// TIA Portal project "Delta_191206" (V15)

(* hardware
DEVICE "S7-1200 station_1"  S7-1200 Station
   slot 0: "Rack_0"  S7-1200 Rack  Rack  V1.0
   slot 1: "PLC_1"  CPU 1215C DC/DC/DC  6ES7 215-1AG40-0XB0  V4.2
   slot 2: "DQ 16x24VDC_1"  6ES7 222-1BH30-0XB0  V1.0
DEVICE "PC station"  SIMATIC PC station
   slot 0: "PC station"  Rail  SIMATIC PC-Station  V1.0
      slot 125: "Stationmanager"  Station_Manager  V6.0.4
   slot 1: "IE general"  IE General  IE_CP  V8.2.0
   slot 2: "OPC Server_1"  OPC Server  OPC Server  V8.2.0
*)

// ===== PLC "PLC_1"  CPU 1215C DC/DC/DC =====

VAR_GLOBAL   // PLC tag table "Default tag table"
   "start" AT %I0.2 : Bool;
   "stop" AT %I0.3 : Bool;
   "AX_1_Homing switch" AT %I1.2 : Bool;
   "Ready" AT %I0.5 : Bool;
   "Emergency_Stop" AT %I0.7 : Bool;
   "AX_2_Homing switch" AT %I1.1 : Bool;
   "Home" AT %I0.4 : Bool;
   "AX_3_Homing switch" AT %I1.3 : Bool;
   "Tag_13" AT %I0.0 : Bool;
   "Tag_14" AT %I0.1 : Bool;
   "AX_1_Pulse" AT %Q0.0 : Bool;
   "AX_1_Direction" AT %Q0.3 : Bool;
   "AX_1_DriveEnable" AT %Q0.6 : Bool;
   "AX_2_Pulse" AT %Q0.1 : Bool;
   "AX_2_Direction" AT %Q0.4 : Bool;
   "AX_2_DriveEnable" AT %Q0.7 : Bool;
   "AX_3_Direction" AT %Q0.5 : Bool;
   "AX_3_Pulse" AT %Q0.2 : Bool;
   "AX_3_DriveEnable" AT %Q1.0 : Bool;
   "Sys_Start" AT %M0.0 : Bool;
   "tr_0" AT %M1.0 : Bool;
   "pos_on" AT %M2.0 : Bool;
   "AX_1_done" AT %M3.0 : Bool;
   "AX_2_done" AT %M3.1 : Bool;
   "AX_3_done" AT %M3.2 : Bool;
   "done_1" AT %M3.3 : Bool;
   "done_2" AT %M3.4 : Bool;
   "done_3" AT %M3.5 : Bool;
   "ind" AT %MW4 : Int;
   "tr_1" AT %M1.1 : Bool;
   "tr_3" AT %M1.3 : Bool;
   "tr_4" AT %M1.4 : Bool;
   "tr_5" AT %M1.5 : Bool;
   "tr_6" AT %M1.6 : Bool;
   "Tag_8" AT %M0.1 : Bool;
   "Tag_9" AT %M0.2 : Bool;
   "tr_7" AT %M1.7 : Bool;
   "tr_2" AT %M1.2 : Bool;
   "Tag_3" AT %M2.2 : Bool;
   "Tag_4" AT %M2.1 : Bool;
   "Tag_5" AT %M2.3 : Bool;
   "Tag_6" AT %M2.4 : Bool;
   "home_ypd" AT %M2.5 : Bool;
   "Tag_2" AT %MD6 : Real;
   "Tag_10" AT %MD10 : Real;
   "Tag_11" AT %MD14 : Real;
   "Tag_12" AT %MD20 : Real;
   "Tag_15" AT %M20.0 : Bool;
   "Tag_16" AT %M2.7 : Bool;
   "Tag_17" AT %M20.3 : Bool;
   "Tag_18" AT %M20.4 : Bool;
   "Tag_19" AT %M20.5 : Bool;
   "Tag_20" AT %M20.1 : Bool;
   "Tag_21" AT %M20.2 : Bool;
   "Tag_22" AT %M20.6 : Bool;
   "Tag_23" AT %M20.7 : Bool;
   "Tag_7" AT %M21.0 : Bool;
   "vakum" AT %Q1.1 : Bool;
   "Tag_25" AT %M4.0 : Bool;
   "Tag_26" AT %M22.0 : Bool;
   "Reset" AT %I0.6 : Bool;
   "gui_start" AT %M23.0 : Bool;
   "gui_stop" AT %M23.1 : Bool;
   "gui_homing" AT %M23.2 : Bool;
   "gui_startpackaging" AT %M23.3 : Bool;
   "gui_reset" AT %M23.4 : Bool;
END_VAR

DATA_BLOCK "OPC_DATA"   // DB5
{ S7_Optimized_Access := 'FALSE' }
VERSION : 0.1
   VAR
      x1_pos : Array[0..100] of Real;
      x2_pos : Array[0..100] of Real;
      x3_pos : Array[0..100] of Real;
      x1_vlcty : Array[0..100] of Real;
      x2_vlcty : Array[0..100] of Real;
      x3_vlcty : Array[0..100] of Real;
      manuel_array : Array[0..100] of Int;
      vakum : Array[0..100] of Int;
   END_VAR
BEGIN
   x1_pos[1] := 0.0;
   x1_pos[0] := 0.0;
   x2_pos[0] := 0.0;
   x2_pos[1] := 0.0;
   x3_pos[0] := 0.0;
   x3_pos[1] := 0.0;
   x1_pos[2] := 0.0;
END_DATA_BLOCK

DATA_BLOCK "AX_1"   // DB1, Motion_DB
{ S7_Optimized_Access := 'TRUE' }
AUTHOR : SIMATIC
FAMILY : BasicMC
NAME : TO_PosAx
VERSION : 6.0
// stored: InstanceOfName TO_PositioningAxis
"TO_PositioningAxis"
BEGIN
   // Axis.HomingReferencePointSwitch_AddressCU = %I1.2
   // Axis.EnableOutput_AddressCU = %Q0.6
   // Axis.DirectionOutputEnabledCU = TRUE
   // Axis.OnlinePtoModeCU = 16#0000_0002
   // Axis.SelectedChannel2EnumCU = %Q0.3
   // Axis.SelectedChannel1EnumCU = %Q0.0
   // Pulse.MinDeltaDeltaFrequencyCU = 0.004
   // Pulse.MaxDeltaDeltaFrequencyCU = 1.0E+10
   // Pulse.MinDeltaFrequencyCU = 0.005
   // Pulse.MaxDeltaFrequencyCU = 9.5E+9
   // Pulse.MinFrequencyCU = 1.0
   // Pulse.MaxFrequencyCU = 100000.0
   // Pulse.OutputSourceCU = 16#0000_0000
   // Axis.SelectPTO = 0
END_DATA_BLOCK

DATA_BLOCK "AX_2"   // DB2, Motion_DB
{ S7_Optimized_Access := 'TRUE' }
AUTHOR : SIMATIC
FAMILY : BasicMC
NAME : TO_PosAx
VERSION : 6.0
// stored: InstanceOfName TO_PositioningAxis
"TO_PositioningAxis"
BEGIN
   // Axis.HomingReferencePointSwitch_AddressCU = %I1.1
   // Axis.EnableOutput_AddressCU = %Q0.7
   // Axis.DirectionOutputEnabledCU = TRUE
   // Axis.OnlinePtoModeCU = 16#0000_0002
   // Axis.SelectedChannel2EnumCU = %Q0.4
   // Axis.SelectedChannel1EnumCU = %Q0.1
   // Pulse.MinDeltaDeltaFrequencyCU = 0.004
   // Pulse.MaxDeltaDeltaFrequencyCU = 1.0E+10
   // Pulse.MinDeltaFrequencyCU = 0.005
   // Pulse.MaxDeltaFrequencyCU = 9.5E+9
   // Pulse.MinFrequencyCU = 1.0
   // Pulse.MaxFrequencyCU = 100000.0
   // Pulse.OutputSourceCU = 16#0000_0000
   // Axis.SelectPTO = 1
   // Axis.OnlinePtoIndexCU = 1
END_DATA_BLOCK

DATA_BLOCK "AX_3"   // DB3, Motion_DB
{ S7_Optimized_Access := 'TRUE' }
AUTHOR : SIMATIC
FAMILY : BasicMC
NAME : TO_PosAx
VERSION : 6.0
// stored: InstanceOfName TO_PositioningAxis
"TO_PositioningAxis"
BEGIN
   // Axis.HomingReferencePointSwitch_AddressCU = %I1.3
   // Axis.EnableOutput_AddressCU = %Q1.0
   // Axis.DirectionOutputEnabledCU = TRUE
   // Axis.OnlinePtoModeCU = 16#0000_0002
   // Axis.SelectedChannel2EnumCU = %Q0.5
   // Axis.SelectedChannel1EnumCU = %Q0.2
   // Pulse.MinDeltaDeltaFrequencyCU = 0.004
   // Pulse.MaxDeltaDeltaFrequencyCU = 1.0E+10
   // Pulse.MinDeltaFrequencyCU = 0.005
   // Pulse.MaxDeltaFrequencyCU = 9.5E+9
   // Pulse.MinFrequencyCU = 1.0
   // Pulse.MaxFrequencyCU = 100000.0
   // Pulse.OutputSourceCU = 16#0000_0000
   // Axis.SelectPTO = 2
   // Axis.OnlinePtoIndexCU = 2
END_DATA_BLOCK

ORGANIZATION_BLOCK "Main"   // OB1, LAD, ProgramCycle
TITLE = "Main Program Sweep (Cycle)"
{ S7_Optimized_Access := 'TRUE' }
VERSION : 0.1
   VAR_INPUT
      Initial_Call : Bool;   // Initial call of this OB
      Remanence : Bool;   // =True, if remanent data are available
   END_VAR
   VAR_TEMP   // added for the SCL form of the ladder/FBD networks
      _w1 : Bool;
      _w2 : Bool;
      _w3 : Bool;
   END_VAR
BEGIN

REGION Network 1: HALT
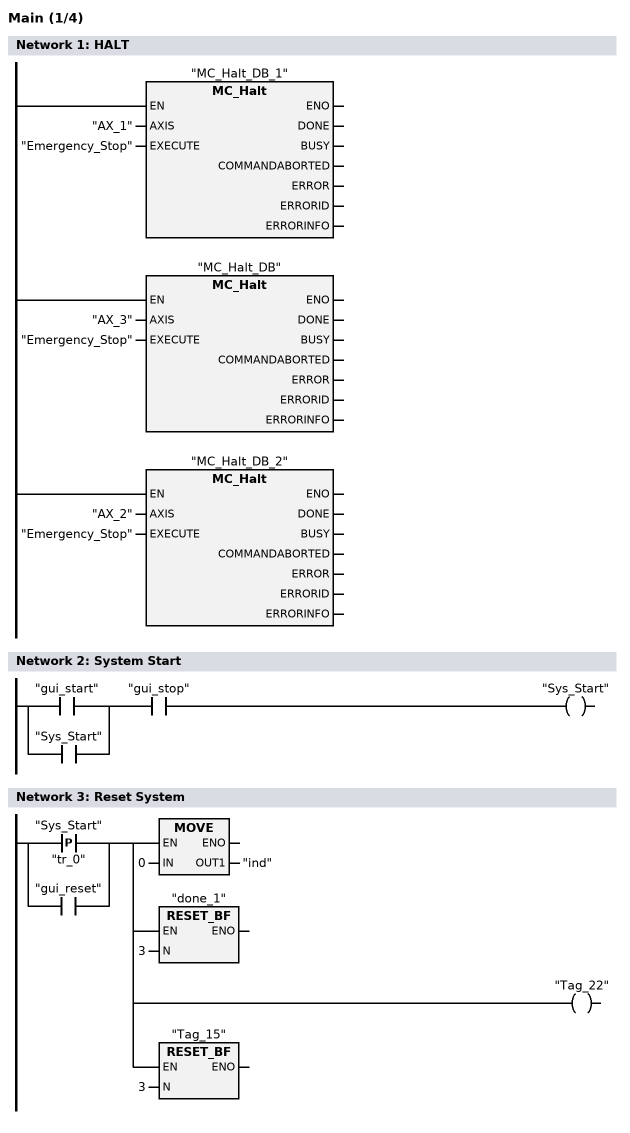
   "MC_Halt_DB_1"(Axis := "AX_1", Execute := "Emergency_Stop");   // MC_Halt
   "MC_Halt_DB"(Axis := "AX_3", Execute := "Emergency_Stop");   // MC_Halt
   "MC_Halt_DB_2"(Axis := "AX_2", Execute := "Emergency_Stop");   // MC_Halt
END_REGION

REGION Network 2: System Start
   RUNG wire#powerrail
      Contact( "gui_start" )
      wire#w1
      Contact( "gui_stop" )
      Coil( "Sys_Start" )
   END_RUNG
   RUNG wire#powerrail
      Contact( "Sys_Start" )
   END_RUNG wire#w1
   // the same network as SCL:
   "Sys_Start" := ("gui_start" OR "Sys_Start") AND "gui_stop";
END_REGION

REGION Network 3: Reset System
   // no SCL statement known for RBitfield: written as a call
   #_w1 := "Sys_Start" AND NOT "tr_0";   // rising edge of "Sys_Start"
   "tr_0" := "Sys_Start";
   #_w2 := #_w1 OR "gui_reset";
   IF #_w2 THEN
       "ind" := 0;
       RESET_BF(operand := "done_1", n := 3);
   END_IF;
   "Tag_22" := #_w2;
   IF #_w2 THEN RESET_BF(operand := "Tag_15", n := 3); END_IF;
END_REGION

REGION Network 4: Motor Enable
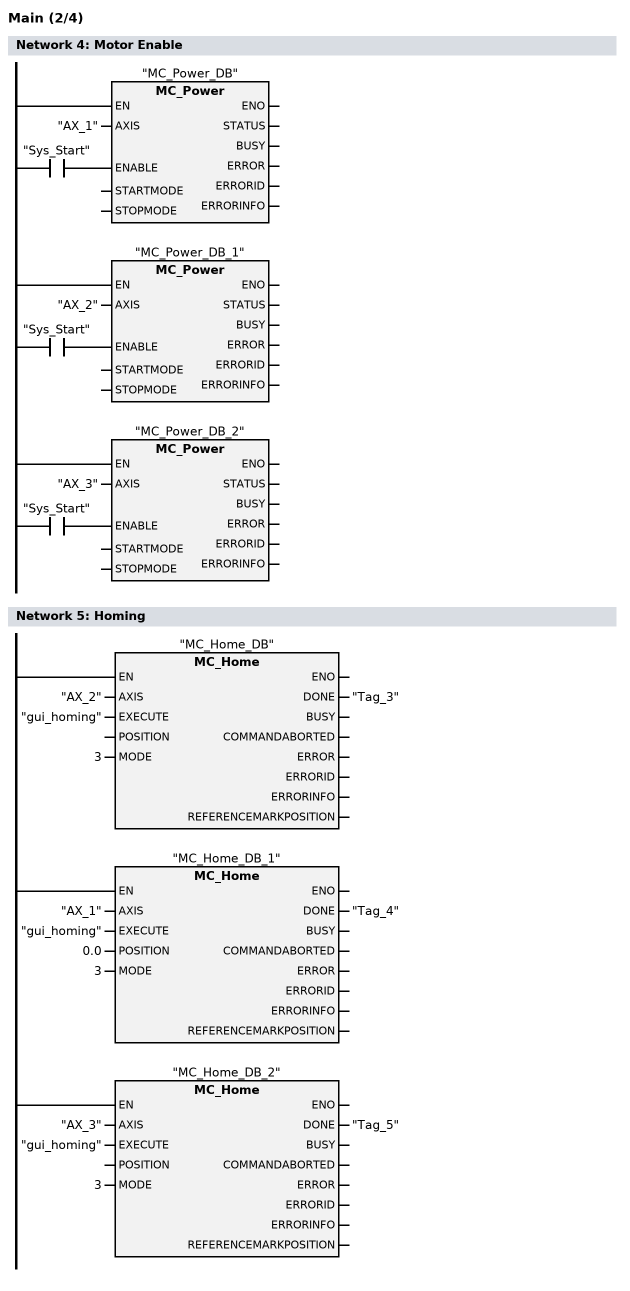
   "MC_Power_DB"(Axis := "AX_1", Enable := "Sys_Start");   // MC_Power
   "MC_Power_DB_1"(Axis := "AX_2", Enable := "Sys_Start");   // MC_Power
   "MC_Power_DB_2"(Axis := "AX_3", Enable := "Sys_Start");   // MC_Power
END_REGION

REGION Network 5: Homing
   "MC_Home_DB"(Axis := "AX_2", Execute := "gui_homing", Mode := 3, Done => "Tag_3");   // MC_Home
   "MC_Home_DB_1"(Axis := "AX_1", Execute := "gui_homing", Position := 0.0, Mode := 3, Done => "Tag_4");   // MC_Home
   "MC_Home_DB_2"(Axis := "AX_3", Execute := "gui_homing", Mode := 3, Done => "Tag_5");   // MC_Home
END_REGION

REGION Network 6: Home and Done Bit Data Saved
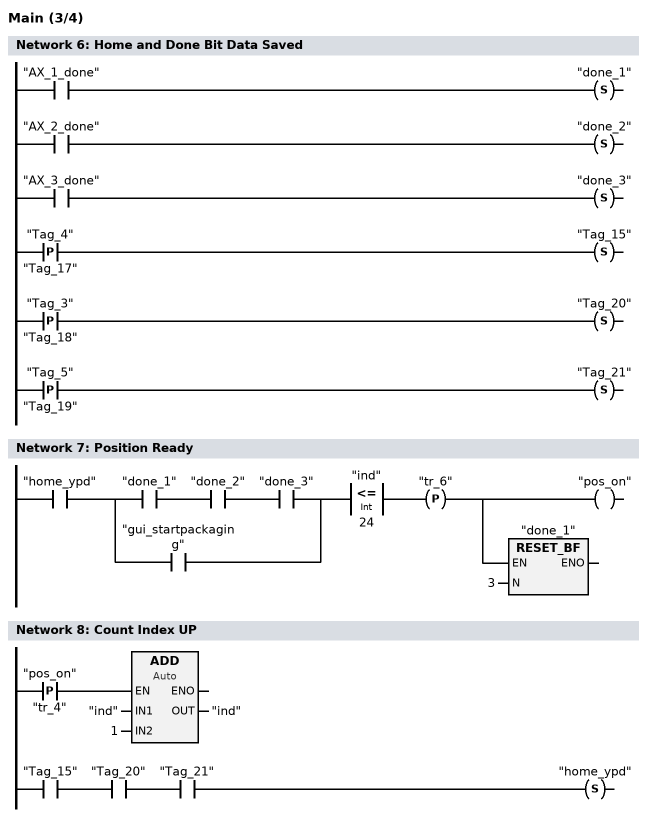
   RUNG wire#powerrail
      Contact( "AX_1_done" )
      S_Coil( "done_1" )
   END_RUNG
   RUNG wire#powerrail
      Contact( "AX_2_done" )
      S_Coil( "done_2" )
   END_RUNG
   RUNG wire#powerrail
      Contact( "AX_3_done" )
      S_Coil( "done_3" )
   END_RUNG
   RUNG wire#powerrail
      P_Contact(operand := "Tag_4", bit := "Tag_17")
      S_Coil( "Tag_15" )
   END_RUNG
   RUNG wire#powerrail
      P_Contact(operand := "Tag_3", bit := "Tag_18")
      S_Coil( "Tag_20" )
   END_RUNG
   RUNG wire#powerrail
      P_Contact(operand := "Tag_5", bit := "Tag_19")
      S_Coil( "Tag_21" )
   END_RUNG
   // the same network as SCL:
   IF "AX_1_done" THEN "done_1" := TRUE; END_IF;
   IF "AX_2_done" THEN "done_2" := TRUE; END_IF;
   IF "AX_3_done" THEN "done_3" := TRUE; END_IF;
   #_w1 := "Tag_4" AND NOT "Tag_17";   // rising edge of "Tag_4"
   "Tag_17" := "Tag_4";
   IF #_w1 THEN "Tag_15" := TRUE; END_IF;
   #_w2 := "Tag_3" AND NOT "Tag_18";   // rising edge of "Tag_3"
   "Tag_18" := "Tag_3";
   IF #_w2 THEN "Tag_20" := TRUE; END_IF;
   #_w3 := "Tag_5" AND NOT "Tag_19";   // rising edge of "Tag_5"
   "Tag_19" := "Tag_5";
   IF #_w3 THEN "Tag_21" := TRUE; END_IF;
END_REGION

REGION Network 7: Position Ready
   // no SCL statement known for RBitfield: written as a call
   #_w1 := "home_ypd" AND (("done_1" AND "done_2" AND "done_3") OR "gui_startpackaging") AND ("ind" <= 24);
   #_w2 := #_w1 AND NOT "tr_6";   // rising edge
   "tr_6" := #_w1;
   "pos_on" := #_w2;
   IF #_w2 THEN RESET_BF(operand := "done_1", n := 3); END_IF;
END_REGION

REGION Network 8: Count Index UP
   RUNG wire#powerrail
      P_Contact(operand := "pos_on", bit := "tr_4")
      Add(in1 := "ind", in2 := 1, out => "ind")
   END_RUNG
   RUNG wire#powerrail
      Contact( "Tag_15" )
      Contact( "Tag_20" )
      Contact( "Tag_21" )
      S_Coil( "home_ypd" )
   END_RUNG
   // the same network as SCL:
   #_w1 := "pos_on" AND NOT "tr_4";   // rising edge of "pos_on"
   "tr_4" := "pos_on";
   IF #_w1 THEN "ind" := "ind" + 1; END_IF;
   IF "Tag_15" AND "Tag_20" AND "Tag_21" THEN "home_ypd" := TRUE; END_IF;
END_REGION

REGION Network 9: Move Motors
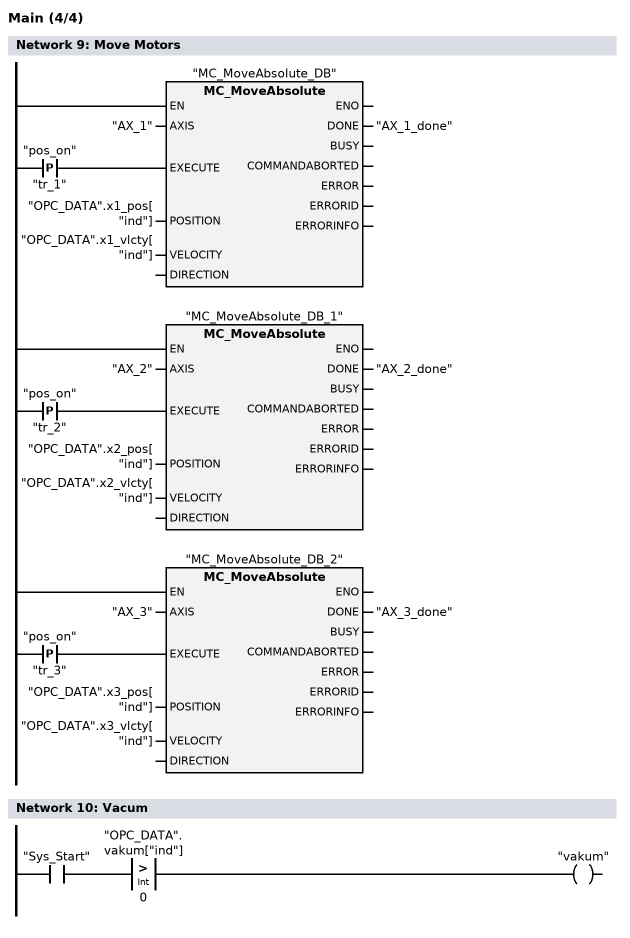
   #_w1 := "pos_on" AND NOT "tr_1";   // rising edge of "pos_on"
   "tr_1" := "pos_on";
   "MC_MoveAbsolute_DB"(Axis := "AX_1",   // MC_MoveAbsolute
                        Execute := #_w1,
                        Position := "OPC_DATA".x1_pos["ind"],
                        Velocity := "OPC_DATA".x1_vlcty["ind"],
                        Done => "AX_1_done");
   #_w2 := "pos_on" AND NOT "tr_2";   // rising edge of "pos_on"
   "tr_2" := "pos_on";
   "MC_MoveAbsolute_DB_1"(Axis := "AX_2",   // MC_MoveAbsolute
                          Execute := #_w2,
                          Position := "OPC_DATA".x2_pos["ind"],
                          Velocity := "OPC_DATA".x2_vlcty["ind"],
                          Done => "AX_2_done");
   #_w3 := "pos_on" AND NOT "tr_3";   // rising edge of "pos_on"
   "tr_3" := "pos_on";
   "MC_MoveAbsolute_DB_2"(Axis := "AX_3",   // MC_MoveAbsolute
                          Execute := #_w3,
                          Position := "OPC_DATA".x3_pos["ind"],
                          Velocity := "OPC_DATA".x3_vlcty["ind"],
                          Done => "AX_3_done");
END_REGION

REGION Network 10: Vacum
   RUNG wire#powerrail
      Contact( "Sys_Start" )
      { S7_Templates := "SrcType := Int" } GT_Contact(in1 := "OPC_DATA".vakum["ind"], in2 := 0)
      Coil( "vakum" )
   END_RUNG
   // the same network as SCL:
   "vakum" := "Sys_Start" AND ("OPC_DATA".vakum["ind"] > 0);
END_REGION
END_ORGANIZATION_BLOCK